// Mitsubishi GX Works2 project: 2023-06-19 #1 생산자동화기능사 18번   PLC: Q03UDV
// 생산자동화기능사

// global labels: Global1
VAR_GLOBAL
  PB1 AT X0 : BOOL;
  PB2 AT X1 : BOOL;
  정지 AT X2 : BOOL;
  공급후진 AT X3 : BOOL;
  공급전진 AT X4 : BOOL;
  가공후진 AT X5 : BOOL;
  가공전진 AT X6 : BOOL;
  송출후진 AT X7 : BOOL;
  송출전진 AT X8 : BOOL;
  배출후진 AT X9 : BOOL;
  배출전진 AT X0A : BOOL;
  매거진 AT X0B : BOOL;
  금속센서 AT X0F : BOOL;
  PB3 AT X0C : BOOL;
  적색 AT Y20 : BOOL;
  황색 AT Y21 : BOOL;
  녹색 AT Y22 : BOOL;
  공급1 AT Y23 : BOOL;
  공급2 AT Y24 : BOOL;
  가공 AT Y25 : BOOL;
  드릴 AT Y26 : BOOL;
  송출 AT Y27 : BOOL;
  배출 AT Y28 : BOOL;
  컨베이어 AT Y29 : BOOL;
END_VAR

PROGRAM 테스트동작
VAR
  PHASE : INT;
END_VAR
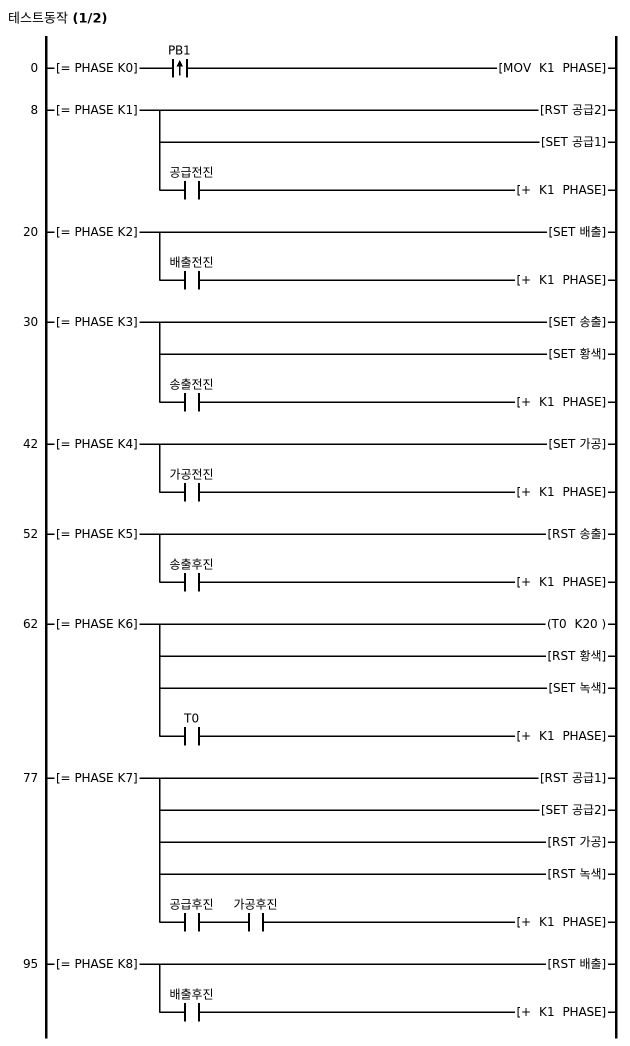
0     LD=     PHASE K0
      ANDP    PB1
      MOV     K1 PHASE
8     LD=     PHASE K1
      RST     공급2
      SET     공급1
      AND     공급전진
      +       K1 PHASE
20    LD=     PHASE K2
      SET     배출
      AND     배출전진
      +       K1 PHASE
30    LD=     PHASE K3
      SET     송출
      SET     황색
      AND     송출전진
      +       K1 PHASE
42    LD=     PHASE K4
      SET     가공
      AND     가공전진
      +       K1 PHASE
52    LD=     PHASE K5
      RST     송출
      AND     송출후진
      +       K1 PHASE
62    LD=     PHASE K6
      OUT     T0 K20
      RST     황색
      SET     녹색
      AND     T0
      +       K1 PHASE
77    LD=     PHASE K7
      RST     공급1
      SET     공급2
      RST     가공
      RST     녹색
      AND     공급후진
      AND     가공후진
      +       K1 PHASE
95    LD=     PHASE K8
      RST     배출
      AND     배출후진
      +       K1 PHASE
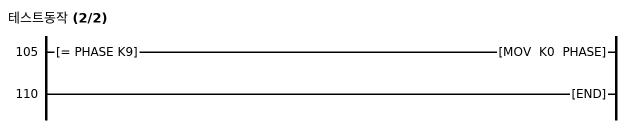
105   LD=     PHASE K9
      MOV     K0 PHASE
110   END
END_PROGRAM

PROGRAM 생산자동화기능사
VAR
  PHASE : INT;
  MODE : INT;
END_VAR
VAR CONSTANT
  단속 : INT;
  연속 : INT := 1;
END_VAR
VAR
  METAL : INT;
  NMETAL : INT;
  BLINK1 : ARRAY [0..3] OF BOOL;
  BLINK2 : ARRAY [0..3] OF BOOL;
  QUIT : BOOL;
  EMG : INT;
  BLINK3 : ARRAY [0..3] OF BOOL;
END_VAR
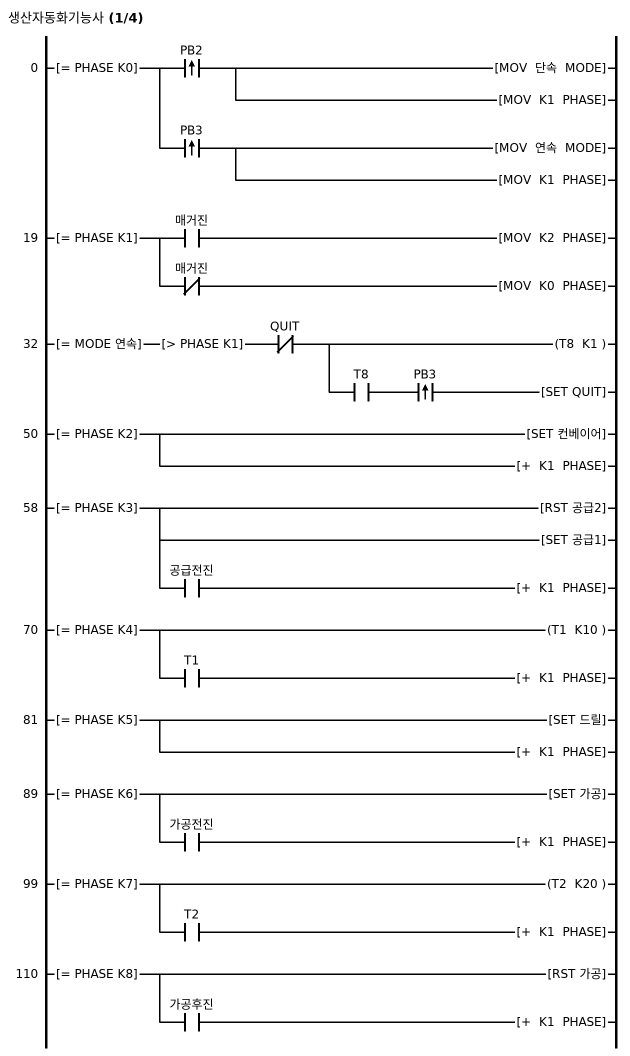
0     LD=     PHASE K0
      MPS
      ANDP    PB2
      MOV     단속 MODE
      MOV     K1 PHASE
      MPP
      ANDP    PB3
      MOV     연속 MODE
      MOV     K1 PHASE
19    LD=     PHASE K1
      MPS
      AND     매거진
      MOV     K2 PHASE
      MPP
      ANI     매거진
      MOV     K0 PHASE
32    LD=     MODE 연속
      AND>    PHASE K1
      ANI     QUIT
      OUT     T8 K1
      AND     T8
      ANDP    PB3
      SET     QUIT
50    LD=     PHASE K2
      SET     컨베이어
      +       K1 PHASE
58    LD=     PHASE K3
      RST     공급2
      SET     공급1
      AND     공급전진
      +       K1 PHASE
70    LD=     PHASE K4
      OUT     T1 K10
      AND     T1
      +       K1 PHASE
81    LD=     PHASE K5
      SET     드릴
      +       K1 PHASE
89    LD=     PHASE K6
      SET     가공
      AND     가공전진
      +       K1 PHASE
99    LD=     PHASE K7
      OUT     T2 K20
      AND     T2
      +       K1 PHASE
110   LD=     PHASE K8
      RST     가공
      AND     가공후진
      +       K1 PHASE
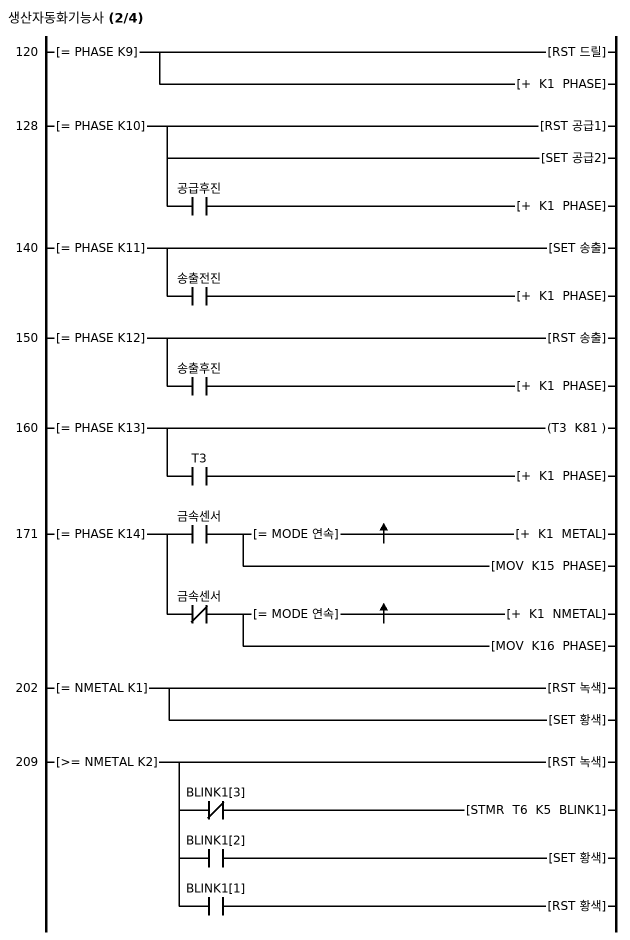
120   LD=     PHASE K9
      RST     드릴
      +       K1 PHASE
128   LD=     PHASE K10
      RST     공급1
      SET     공급2
      AND     공급후진
      +       K1 PHASE
140   LD=     PHASE K11
      SET     송출
      AND     송출전진
      +       K1 PHASE
150   LD=     PHASE K12
      RST     송출
      AND     송출후진
      +       K1 PHASE
160   LD=     PHASE K13
      OUT     T3 K81
      AND     T3
      +       K1 PHASE
171   LD=     PHASE K14
      MPS
      AND     금속센서
      MPS
      AND=    MODE 연속
      MEP
      +       K1 METAL
      MPP
      MOV     K15 PHASE
      MPP
      ANI     금속센서
      MPS
      AND=    MODE 연속
      MEP
      +       K1 NMETAL
      MPP
      MOV     K16 PHASE
202   LD=     NMETAL K1
      RST     녹색
      SET     황색
209   LD>=    NMETAL K2
      RST     녹색
      MPS
      ANI     BLINK1[3]
      STMR    T6 K5 BLINK1
      MRD
      AND     BLINK1[2]
      SET     황색
      MPP
      AND     BLINK1[1]
      RST     황색
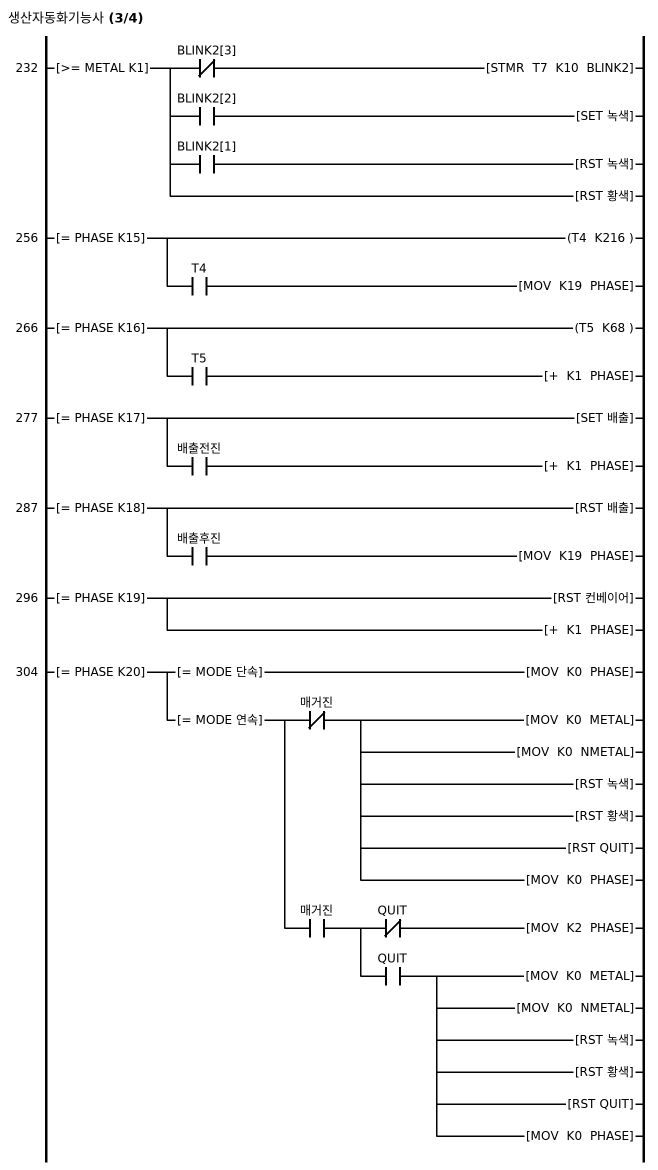
232   LD>=    METAL K1
      MPS
      ANI     BLINK2[3]
      STMR    T7 K10 BLINK2
      MRD
      AND     BLINK2[2]
      SET     녹색
      MRD
      AND     BLINK2[1]
      RST     녹색
      MPP
      RST     황색
256   LD=     PHASE K15
      OUT     T4 K216
      AND     T4
      MOV     K19 PHASE
266   LD=     PHASE K16
      OUT     T5 K68
      AND     T5
      +       K1 PHASE
277   LD=     PHASE K17
      SET     배출
      AND     배출전진
      +       K1 PHASE
287   LD=     PHASE K18
      RST     배출
      AND     배출후진
      MOV     K19 PHASE
296   LD=     PHASE K19
      RST     컨베이어
      +       K1 PHASE
304   LD=     PHASE K20
      MPS
      AND=    MODE 단속
      MOV     K0 PHASE
      MPP
      AND=    MODE 연속
      MPS
      ANI     매거진
      MOV     K0 METAL
      MOV     K0 NMETAL
      RST     녹색
      RST     황색
      RST     QUIT
      MOV     K0 PHASE
      MPP
      AND     매거진
      MPS
      ANI     QUIT
      MOV     K2 PHASE
      MPP
      AND     QUIT
      MOV     K0 METAL
      MOV     K0 NMETAL
      RST     녹색
      RST     황색
      RST     QUIT
      MOV     K0 PHASE
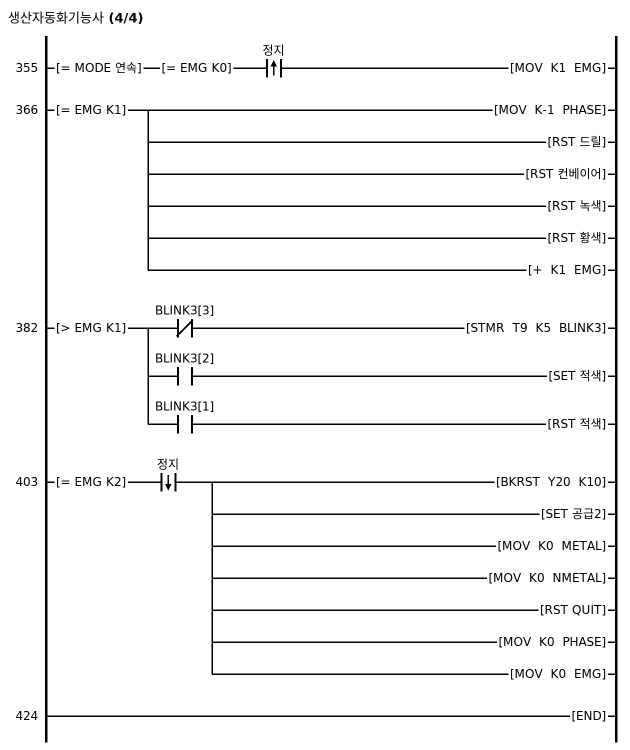
355   LD=     MODE 연속
      AND=    EMG K0
      ANDP    정지
      MOV     K1 EMG
366   LD=     EMG K1
      MOV     K-1 PHASE
      RST     드릴
      RST     컨베이어
      RST     녹색
      RST     황색
      +       K1 EMG
382   LD>     EMG K1
      MPS
      ANI     BLINK3[3]
      STMR    T9 K5 BLINK3
      MRD
      AND     BLINK3[2]
      SET     적색
      MPP
      AND     BLINK3[1]
      RST     적색
403   LD=     EMG K2
      ANDF    정지
      BKRST   Y20 K10
      SET     공급2
      MOV     K0 METAL
      MOV     K0 NMETAL
      RST     QUIT
      MOV     K0 PHASE
      MOV     K0 EMG
424   END
END_PROGRAM
